// TIA Portal V19 export
TYPE "FsCore"
// stored: Access Published
   STRUCT
      OKTAG : Bool := FALSE;
      HomePos : LReal := 0.0;   // GoHome target position [Axis UM]
      HomeVelocity : LReal;   // Return velocity [Axis UM]
      Acc : LReal;
      Jerk : LReal;
      ErrWindow : LReal;
      ErrDwellTime : Time;
      ErrTimeout : Time;
      FAK : LReal := 1.0;   // FAK material to axis ratio
      AxMODULO : LReal := 0.0;
      MasterPosition : LReal;   // Actual position of Lead axis
      SlavePosition : LReal;   // Actual Position of Follower axis
      MaterialPosition : LReal;   // Lead/following relative position
      MasterVelocity : LReal;   // Velocity of lead axis
      StartAdvance : LReal;   // Advance space
      SyncDelay : LReal;
      MasterExtraSpeed : Real;   // Extra-velocity
      SlaveVelocity : LReal;   // Velocity of following axis
      SlaveAcceleration : LReal;   // Actual Following axis Acceleration
      WorkPosition : LReal;   // Work Position
      Fct : UInt;   // Flying shear phase
      Sts : Struct   // Status
         Standstill : Bool;   // Following axis standstill
         NotReachable : Bool;   // Work position not reachable
         NotSynched : Bool;   // Work position not synched
         ErrTimeout : Bool;   // Work command on timeout
         NotPermitted : Bool;   // Procedure aborted cause of missed permission
      END_STRUCT;
      iWorkPosition : LReal;   // Internal work position
      iSlaveSynchPos : LReal;
      iMasterSyncPos : LReal;
      iStartTrigger : Bool := FALSE;
      iSpaceToGo : LReal;
      iMasterSynchSpace : LReal;
      iSlaveSynchSpace : LReal;
      iMasterLag : LReal;   // Missing space to synchro position
      iJerkToUse : LReal;   // Jerk to use
      "K_mV_TO_m/s" : LReal;   // from lead Velocity UM to m/s
      "K_mA_TO_m/s^2" : LReal;   // from master Aceleration UM to m/s^2
      "K_sV_TO_m/s" : LReal;   // from follower Velocity UM to m/s
      "K_sA_TO_m/s^2" : LReal;   // from follower Aceleration UM to m/s^2
      "K_m/s^3_TO_sJ" : LReal;   // from m/s^3 to slave Jerk UM
      Par_SI : Struct
         Acc : LReal;   // Acceleration [m/s^2]
         Jerk : LReal;   // Jerk [m/s^3]
      END_STRUCT;
   END_STRUCT;
END_TYPE
